// TIA Portal V21 export
DATA_BLOCK "DB608"   // DB608
TITLE = DB608
AUTHOR : PRECISE
FAMILY : PRECISE
// CIP RECIRCULATION
// stored: AutoNumber false, InstanceOfName FB608, InstanceOfType FB
"FB608"
   // VAR_INPUT
   //    CycleEnable : Bool;
   //    CycleRunning : Bool;
   //    SecPulse : Bool;
   //    AlwaysTrue : Bool;
   //    ActualTemperature : Real;
   //    ParaIn : "RecirculationInputs";
   //    ActualPressure : Real;
   //    ActualConductivity : Real;
   // END_VAR
   // VAR_OUTPUT
   //    Started : Bool;
   //    PressureUtilityValve : Bool;
   //    AlkaliInValve : Bool;
   //    AlkaliPump : Bool;
   //    AcidInValve : Bool;
   //    AcidPump : Bool;
   //    "DosingValve(Cond)" : Bool;
   //    "DosingPump(Cond)" : Bool;
   //    HsbCmd : Bool;
   //    RecPump : Bool;
   //    ParaOut : "RecirculationOutputs";
   //    TimePv : DInt;
   //    StepStatus : String[60];
   // END_VAR
   // VAR_IN_OUT
   //    Over : Bool;
   //    OverTemp : Bool;
   //    ControlStarted : Bool;
   //    TimerPaused : Bool;
   //    PressurePostiveTol : Real;
   //    PressureNegativeTol : Real;
   //    LineValves : Bool;
   //    ActualRepetition : Int;
   //    SetTemperature { ExternalAccessible := 'False'; ExternalVisible := 'False'; ExternalWritable := 'False'} : Real;
   //    SetpH : Real;
   //    SetConductivity : Real;
   //    pHReached : Bool;
   //    ConductivityReached : Bool;
   //    CipSelected : Bool;
   // END_VAR
   // VAR
   //    ValveOnDelayPV : Int;
   //    ValveOffDelayPV : Int;
   //    ValveOnDelayPV_1 : Int;
   //    ValveOffDelayPV_1 : Int;
   //    ValveOnDelayPV_2 : Int;
   //    ValveOffDelayPV_2 : Int;
   //    TempPos : Real;
   //    RE1 : Bool;
   //    StepDelay { S7_SetPoint := 'True'} : "FB110";
   //    RE2 { S7_SetPoint := 'True'} : Bool;
   //    RE3 : Bool;
   //    RE4 : Bool;
   //    RE5 : Bool;
   //    Re6 : Bool;
   //    Re7 : Bool;
   //    "timer" : IEC_TIMER;
   // END_VAR
BEGIN
END_DATA_BLOCK
